Staubli VAL3: GETLINE.pgx

public program GetLine(num x_nFileID (dimensions=1), string& x_sContext (dimensions=1), bool& x_bRes (dimensions=1))
  local num l_nNum
begin


  //文件标志符

  x_bRes=false
  if x_nFileID<0 or x_nFileID>9
    return
  endIf
  //
  switch x_nFileID
    case 0
      l_nNum=$fileGet(0,x_sContext,1)
    break

    case 1
      l_nNum=$fileGet(1,x_sContext,1)
    break

    case 2
      l_nNum=$fileGet(2,x_sContext,1)
    break

    case 3
      l_nNum=$fileGet(3,x_sContext,1)
    break

    case 4
      l_nNum=$fileGet(4,x_sContext,1)
    break

    case 5
      l_nNum=$fileGet(5,x_sContext,1)
    break
    case 6
      l_nNum=$fileGet(6,x_sContext,1)
    break

    case 7
      l_nNum=$fileGet(7,x_sContext,1)
    break
    case 8
      l_nNum=$fileGet(8,x_sContext,1)
    break

    case 9
      l_nNum=$fileGet(9,x_sContext,1)
    break


  endSwitch
  if l_nNum!=1
    return
  endIf
  x_bRes=true




end
